PROGRAM P_Set_Research_Data
VAR
END_VAR

//***********************************************************************************
//
// ETH Zürich / Robotic Fabrication Lab
// HIB C 13 / Stefano-Franscini-Platz 1
// CH-8093 Zürich
// 
// ***********************************************************************************
// 
// PROJECT     :  A061 Inline Mixer
// 
// FUNCTION    :  Set all research data for the process
// 
// AUTHOR      :  Seyma Gürel / Philippe Fleischmann / Weiting Chen
// 
// EMAIL       :  scotto@arch.ethz.ch / fleischmann@arch.ehtz.ch
// 
// Copyright   :  ETH Zürich (CH) 2022
//
// ***********************************************************************************


//***********************************************************************************
// Inline mixer 
//***********************************************************************************

// Updating Mixer 1 max speed
GVL_VAR.f_MI1_MaxSpeed:= 720; // [distance/s] ( equel to 120 rpm, by measurement 221006)



//***********************************************************************************
// Superplasticizer pump 
//***********************************************************************************

// Updating Superplasticizer Pump checking values (WT
GVL_ResearchData.n_RED_Superplasticizer_Pump_Check_Flowrate:=9;           // [ml/min]
GVL_ResearchData.n_RED_Superplasticizer_Pump_Check_Duration:=T#60000MS;   // [ms]
//GVL_ResearchData.f_RED_Superplasticizer_Pump_Density:=1.06;               // [g/cm^3]

GVL_ResearchData.n_RED_Superplasticizer_Pump_Flush_Flowrate:=GVL_ResearchData.f_RED_Status_Superplasticizer_Pump_Max_Flowrate_ml_per_min;	// [ml/min]
//[32767 is equal 10v output and it means maximum setup speed from ViscoTech 654 rpm]


//***********************************************************************************
// Accelerator pump 1
//***********************************************************************************
//
// Updating Acceleration Pump checking values (WT 
GVL_ResearchData.n_RED_Acceleration_Pump_Check_Flowrate:=90;     		// [ml/min]
GVL_ResearchData.n_RED_Acceleration_Pump_Check_Duration:=T#60000MS;   	// [ms]
//GVL_ResearchData.f_RED_Acceleration_Pump_Density:=1.62;               // [kg/m^3]
GVL_ResearchData.n_RED_Acceleration_Pump_Flush_Flowrate:=GVL_ResearchData.f_RED_Status_Acceleration_Pump_Max_Flowrate_ml_per_min;	// [ml/min]
//[32767 is equal 10v output and it means maximum setup speed from ViscoTech ? rpm]
GVL_ResearchData.f_RED_Acceleration_Pump_Mass:= (GVL_ResearchData.n_RED_Acceleration_Pump_Check_Flowrate*
												(TO_REAL(GVL_ResearchData.n_RED_Acceleration_Pump_Check_Duration)/TO_REAL(T#60000MS))*
												GVL_ResearchData.f_RED_Acceleration_Pump_Density);



//***********************************************************************************
// Concrete pump 1
//***********************************************************************************
GVL_ResearchData.f_RED_Concrete_Pump_Check_Flowrate:=2.5;		//[l/min] (1.3 to 3.7)
GVL_ResearchData.n_RED_Concrete_Pump_Check_Duration_Time:=T#15000MS;		// [ms]
GVL_ResearchData.n_RED_Concrete_Pump_Flush_Flowrate:=GVL_ResearchData.f_RED_Status_Concrete_Pump_Max_Flowrate_l_per_min; // [l/min]

//GVL_ResearchData.f_RED_Concrete_Pump_Density:=2.307;		// [kg/m^3]
GVL_ResearchData.f_RED_Concrete_Pump_Check_Mass:= (GVL_ResearchData.f_RED_Concrete_Pump_Check_Flowrate * 1000 *
												(TO_REAL(GVL_ResearchData.n_RED_Concrete_Pump_Check_Duration_Time)/TO_REAL(T#60000MS))*
												GVL_ResearchData.f_RED_Concrete_Pump_Density);

END_PROGRAM

(* stored: Version 1.1.0.1, ProductVersion 3.1.4024.2
   POU P_Set_Research_Data: Id {773f30f1-b7d3-4c7e-b27f-8d66212207e7}, SpecialFunc None *)
